FUNCTION_BLOCK FB_SortMoverByPos EXTENDS FB_Sort
VAR_INPUT
END_VAR
VAR_OUTPUT
END_VAR
VAR
END_VAR

(* Please override this method so it returns:
* 0 : a == b
*-1 : a < b
* 1 : a > b
* which a and b are the ADDRESS of the 2 elements you want to compare
*)
METHOD Compare : DINT
VAR_INPUT
	a : PVOID;
	b : PVOID;
END_VAR
VAR
    MoverDict_a : MoverDict;
    MoverDict_b : MoverDict;
END_VAR
Tc2_System.MEMCPY(ADR(MoverDict_a), a, SIZEOF(MoverDict));
Tc2_System.MEMCPY(ADR(MoverDict_b), b, SIZEOF(MoverDict));

IF MoverDict_a.MoverPos < MoverDict_b.MoverPos THEN
    Compare := -1;

ELSIF MoverDict_a.MoverPos > MoverDict_b.MoverPos THEN
    Compare := 1;

ELSE
    Compare := 0;

END_IF
END_METHOD

END_FUNCTION_BLOCK

(* stored: Version 1.1.0.1, ProductVersion 3.1.4024.12
   POU FB_SortMoverByPos: Id {3fd8fd2b-e1df-4cfe-bbd2-e923e9027a98}, SpecialFunc None
   Method Compare: Id {230683ba-3804-4771-9d9e-47ab93ee1628} *)
